// TIA Portal V18 export
DATA_BLOCK "BoilerOpModes"   // DB1016
{ S7_Optimized_Access := 'FALSE' }
VERSION : 0.1
// stored: AutoNumber false, DBAccessibleFromOPCUA true, IsOnlyStoredInLoadMemory false, IsWriteProtectedInAS false
   VAR
      OpModes { S7_SetPoint := 'True'} : "UDT_BoilerOpMode";
   END_VAR
BEGIN
END_DATA_BLOCK
